(* IEC 61131-3 sources: process-and-packaging-plant/codesys/sorting-by-weight, 5 files *)

(* ---- GVL_Sort.st ---- *)
{attribute 'qualified_only'}
VAR_GLOBAL
	// Mock Sorting Simulation
	Arrival_Timer : TON;
	Depart_Timer : TON;

	// Process variables
	Box_Present : BOOL; // TRUE when box is at weighing station
	Weight_PV : REAL := 450.0; // Measured weight (grams)
	Weight_Threshold_Low : REAL := 420.0; // Underweight below this
	Weight_Threshold_High : REAL := 480.0; // Overweight above this
	Conveyor_Run : BOOL; // Conveyor Motor Command
	Sort_Actuator : BOOL; // Diverter actuator (TRUE := divert)
	Box_Count : DINT; // Total boxes processed
	Reject_Count : DINT; // Rejected boxes
	ScanTime : REAL := 0.1; // Scan time (secs)

	// Random Weight
	RandSeed : DWORD := 12345;
	Noise : REAL;
	LCG_Multiplier : DWORD := 1664525;
	LCG_Increment : DWORD := 1013904223;
	LCG_Modulus : DWORD := 10000;
END_VAR

(* ---- PLC_PRG.st ---- *)
// 1. Process Simulation (or Factory I/O inputs later)
IF GVL_sort.Simulation_Mode THEN
	PLC_PRG_MockSort();
END_IF

// 2. Alarms (detect abnormal conditions, runs before interlocks so that Downstream_Fault or Box_Jam_Alarms inhibits conveyor)
PLC_PRG_Alarms();

// 3. Interlocks (decide if converter/diverter can run
Interlocks_LD();

// 4. Sorting Sequence (state machine, counters, diverter, runs after Interlocks to keep Sort_Actuator_Enable fresh)
PLC_PRG_SortingSeq();

// 5. Power Layer (monitor equipment health)
PLC_PRG_PowerLayer();

(* ---- PLC_PRG_MockSort.st ---- *)
(* Mock Sorting Simulation
   Generates periodic box arrivals with random wieghts. Sorting logic reacts to Box_Present and Weight_PV.
   This POU is removed/disabled when Factory I/O is connected.

   Box Cycle:
   1 - Every ~4 secs, a box arrives (Box_Present := TRUE)
   2 - A weight is generated (400-50 g range for example)
   3 - After ~3 secs, the box leaves (Box_Present := FALSE) *)

   // Box Arrival Timer fires every 4 secs when no box is present
   GVL_Sort.Arrival_Timer(IN:= NOT GVL_Sort.Box_Present, PT := T#4s);

   IF GVL_Sort.Arrival_Timer.Q AND NOT GVL_Sort.Box_Present THEN
	   GVL_Sort.Box_Present := TRUE;

	   // Generate random weight in 400-500 grange using LCG
	   GVL_Sort.RandSeed := GVL_Sort.RandSeed * GVL_Sort.LCG_Multiplier + GVL_Sort.LCG_Increment;
	   GVL_Sort.Noise := TO_REAL(GVL_Sort.RandSeed MOD GVL_Sort.LCG_Modulus) / TO_REAL(GVL_Sort.LCG_Modulus);
	   GVL_Sort.Weight_PV := 400.0 + (GVL_Sort.Noise * 100.0);
   END_IF

   // Box departure timer : Box leaves after 3 secs
   GVL_Sort.Depart_Timer(IN := GVL_Sort.Box_Present, PT := T#3S);

   IF GVL_Sort.Depart_Timer.Q THEN
	   GVL_Sort.Box_Present := FALSE;
   END_IF

(* ---- PLC_PRG_PowerLayer.st ---- *)
(* Power Layer - Simulated conveyor + Diverter current
   ---------------------------------------------------
   Base Current + Proportional to conveyor running + Diverter actuation + Noise *)

// Effective Load : Conveyor running + Diverter Actuating

(* It simulates the current drawn for conveyor and diverter to monitor, trend, and alarm.
   The load variable is the total mechanical load on the motor circuit*)

GVL_Sort.Load := 0.0;
IF GVL_Sort.Conveyor_Run THEN // Only conveyor runs, main motor draws current
	GVL_Sort.Load := GVL_Sort.Load + 50.0;
END_IF
IF GVL_Sort.Sort_Actuator THEN // Only diverter actuates, solenoid draws current
	GVL_Sort.Load := GVL_Sort.Load + 30.0;
END_IF

// LCG Noise
(* Added for realism, too negligible to require filtering *)
GVL_Sort.RandSeed := GVL_Sort.RandSeed * GVL_Sort.LCG_Multiplier + GVL_Sort.LCG_Increment;
GVL_Sort.Noise := TO_REAL(GVL_Sort.RandSeed MOD GVL_Sort.LCG_Modulus) / TO_REAL(GVL_Sort.LCG_Modulus);
GVL_Sort.Noise := (GVL_Sort.Noise - 0.5) * GVL_Sort.Noise_Amplitude;

// Simulated Current
GVL_Sort.Sim_Current := GVL_Sort.Base_Current + (GVL_Sort.Load * GVL_Sort.Current_Scale_Factor) + GVL_Sort.Noise;

// Overcurrent Alarm
(* It's here and not in alarms because it depends on Sim_Current computed here, a design choice for convenience rather than a strict necessity*)
GVL_Sort.Overcurrent_Alarm := GVL_Sort.Sim_Current > GVL_Sort.Overcurrent_Threshold;

(* ---- PLC_PRG_SortingSeq.st ---- *)
(* State Machine for sorting sequence
   0 : Idle - waiting for a box
   1 : Stabilize - box present, wait for weight to settle (TON)
   2 : Classify - determine if good/reject
   3 : Divert - If reject, actuate the diverter for a fixed time
   4 : Clear - increment counters, wait for the box to leave *)

CASE GVL_Sort.State OF
	0: // IDLE - Waiting for a box
	// Diverters must be off and timers must be reset. Can't stabilize or classify a box that isn't there.
	// This state ends when a new box enters
	GVL_Sort.Sort_Actuator := FALSE;
	GVL_sort.Weight_Stable := FALSE;
	GVL_Sort.Stabilize_Timer(IN := FALSE);
	GVL_Sort.Divert_Timer(IN := FALSE);

	IF GVL_Sort.Box_Present AND NOT GVL_Sort.Prev_Box THEN
		GVL_Sort.State := 1;
	END_IF

	1 : // Stabilize - wait for weight to settle
	// A box just landed on the scale and the reading is bouncing, run a 500 ms timer, which is enough for the weight to settle.
	// This state ends when the 500 ms timer is done
	GVL_Sort.Stabilize_Timer(IN := TRUE, PT := T#500MS);

	IF GVL_Sort.Stabilize_Timer.Q THEN
		GVL_Sort.Weight_Stable := TRUE;
		GVL_Sort.State := 2;
	END_IF

	2 : // Classify - determine underweight/good/overweight
	// Compare weight to thresholds and set the classify_result variable to 0 (good), 1 (under), 2 (over)
	// This state lasts one scan and ends immediately, go to State 3 if reject, State 4 if good

	IF GVL_Sort.Weight_PV < GVL_Sort.Weight_Threshold_Low THEN
		GVL_Sort.Classify_Result := 1; // Underweight
	ELSIF GVL_Sort.Weight_PV > GVL_Sort.Weight_Threshold_High THEN
		GVL_Sort.Classify_Result := 2; // Overweight
	ELSE
		GVL_Sort.Classify_Result := 0; // Good
	END_IF

	IF GVL_Sort.Classify_Result <> 0 THEN
		GVL_Sort.State := 3; // Reject - divert
	ELSE
		GVL_Sort.State := 4; // Good - clear
	END_IF

	3: // Divert - actuate diverter for a fixed time
	// The box is a reject. Push it off with the diverter by setting Sort_Actuator := TRUE and run a 1 sec timer.
	// The diverter must stay on long enough (for a fixed time) to physically push the box off the converter and increment reject_count. One scan is not enough
	// The state ends when the timer is done
		GVL_Sort.Divert_Timer(IN := GVL_Sort.Sort_Actuator_Enable, PT := T#1S);
		// Change : Run the timer not unconditionally, but when actuator is enabled, aka no downstream fault or conveyor running issue, aka also box is present and no box jam alarm

	IF GVL_Sort.Sort_Actuator_Enable THEN
		GVL_Sort.Sort_Actuator := TRUE;
	END_IF

	IF GVL_Sort.Divert_Timer.Q THEN
		GVL_Sort.Sort_Actuator := FALSE;
		GVL_Sort.Reject_Count := GVL_Sort.Reject_Count + 1;
		GVL_Sort.State := 4;
	END_IF

	4 : // Clear - increment counter, wait for the box to leave
	// The box is leaving the station. Increment count and wait for it to be gone
	// The state ends when variable Box_count is FALSE

	// We use a one-shot flag called Count_Done, because Box_Count increments every scan
	// If the box takes 2 seconds to leave and scantime is 100 ms, 20 increments are added where the correct value is one
	// Hence, Count_Done ensures it only increments once
    IF NOT GVL_Sort.Count_Done THEN
        GVL_Sort.Box_Count := GVL_Sort.Box_Count + 1;
        GVL_Sort.Count_Done := TRUE;
    END_IF

    IF NOT GVL_Sort.Box_Present THEN
        GVL_Sort.Count_Done := FALSE;
        GVL_Sort.State := 0;
    END_IF

END_CASE

// Posedge detection for Box_Present (State 0)
GVL_Sort.Prev_Box := GVL_Sort.Box_Present;
